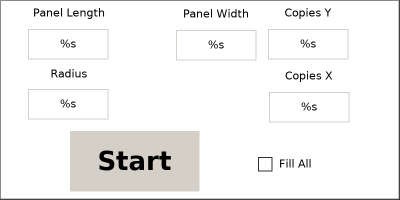
VISUALIZATION V_ProductionMeina2_2Circles  // 400x200
VAR_IN_OUT
	HMI : ST_PackMLBaseModule_HMI;
	HMI_GantryXYZ : ST_GantryXYZ_HMI;
	HMI_Recipe : ST_RecipeBuilder_HMI;
END_VAR
    RoundedRectangle (0,0 400x200)
    RoundedRectangle (70,131 129x60), "Start", colour toggle: HMI.Status.State = E_PMLState.ePMLState_Idle, input disabled if: NOT MAIN.Seedra.RecipeConfig_HMI.Config.IsValid
        OnMouseClick: execute { HMI.Command.State := E_PMLCommand.ePMLCommand_Start; }
    Textfield (28,89 80x30), "%s", text variable: HMI_Recipe.Config.Radius
        OnMouseClick: write the text variable via VisuDialogs.Numpad, min HMI_Recipe.Limits.Radius.MinVal, max HMI_Recipe.Limits.Radius.MaxVal
    Label (11,64 116x20), "Radius"
    Checkbox (256,149 72x30), "Fill All", variable: HMI_Recipe.Config.FillAll
    Textfield (269,92 80x30), "%s", text variable: HMI_Recipe.Config.RequestedCopiesX, input disabled if: MAIN.Seedra.RecipeConfig_HMI.Config.FillAll
        OnMouseClick: write the text variable via VisuDialogs.Numpad, min 1, max MAIN.Seedra.RecipeConfig_HMI.Limits.RequestedCopiesX.MaxVal
    Label (258,66 102x20), "Copies X"
    Textfield (268,29 80x30), "%s", text variable: HMI_Recipe.Config.RequestedCopiesY, input disabled if: MAIN.Seedra.RecipeConfig_HMI.Config.FillAll
        OnMouseClick: write the text variable via VisuDialogs.Numpad, min 1, max MAIN.Seedra.RecipeConfig_HMI.Limits.RequestedCopiesY.MaxVal
    Label (257,3 102x20), "Copies Y"
    Textfield (176,30 80x30), "%s", text variable: HMI_Recipe.Config.PanelFrontWidth
        OnMouseClick: write the text variable via VisuDialogs.Numpad, min HMI_Recipe.Limits.PanelFrontWidth.MinVal, max HMI_Recipe.Limits.PanelFrontWidth.MaxVal
    Textfield (28,29 80x30), "%s", text variable: HMI_Recipe.Config.PanelFrontLength
        OnMouseClick: write the text variable via VisuDialogs.Numpad, min HMI_Recipe.Limits.PanelFrontLength.MinVal, max HMI_Recipe.Limits.PanelFrontLength.MaxVal
    Label (11,3 116x20), "Panel Length"
    Label (127,4 178x20), "Panel Width"
END_VISUALIZATION

(* stored: Version 1.1.0.1, ProductVersion 3.1.4024.15
   Visu V_ProductionMeina2_2Circles: Id {ceb3d707-85b5-4ea5-bea9-aa2192732bf6} *)
